{attribute 'qualified_only'}
VAR_GLOBAL
	Tags: TagsRedundancy;	
END_VAR

(* stored: Version 1.1.0.1, ProductVersion 3.1.4024.6
   GVL GVL_Redundancy: Id {2fc4b88e-b988-4f7a-ac68-f9d0e545a4a6} *)
